FUNCTION_BLOCK FB_TemperatureSensorPCH EXTENDS FB_Sensor
VAR_INPUT
END_VAR
VAR_OUTPUT
	fTemperature : REAL; //measured temperature in °C
END_VAR
VAR
	//I/O-Links
	temperature_IN AT %I* : INT;
	
END_VAR

METHOD GetState_AI : BOOL
VAR_INPUT
END_VAR
fTemperature := temperature_IN*0.1; //conversion

//sensor state
sensorState.fValue := fTemperature;
sensorState.sUnit := 'degreeC';
END_METHOD

END_FUNCTION_BLOCK

(* stored: Version 1.1.0.1, ProductVersion 3.1.4024.6
   POU FB_TemperatureSensorPCH: Id {2248c7c1-cccf-46d0-8556-65f548691921}, SpecialFunc None
   Method GetState_AI: Id {fdfe7e3e-8cc7-4ef0-a7ce-db6d33db1077} *)
